// TIA Portal V20 export
// export: Created 2025-12-01T14:57:17.9653738Z, ExportSetting None, DisplayName Totally Integrated Automation Portal, DisplayVersion V20 Update 3, DisplayName TIA Portal Openness, DisplayVersion V20 Update 3, DisplayName TIA Portal Version Control Interface, DisplayVersion V20 Update 3, DisplayName STEP 7 Professional, DisplayVersion V20 Update 3, DisplayName STEP 7 Safety, DisplayVersion V20 Update 2, DisplayName WinCC Basic/Comfort/Advanced, DisplayVersion V20 Update 3, DisplayName WinCC Professional, DisplayVersion V20 Update 3, DisplayName WinCC Unified, DisplayVersion V20 Update 3
DATA_BLOCK "DB707_JDT02EventosGenerados"   // DB707
{ S7_Optimized_Access := 'FALSE' }
AUTHOR : TRACKING
NAME : 20130301
VERSION : 3.0
// stored: AutoNumber false
   VAR
      Mensaje : Array[0..9999] of Char;
   END_VAR
BEGIN
END_DATA_BLOCK
